{attribute 'qualified_only'}
VAR_GLOBAL
		
	//AnyEstopPressed 			: BOOL;
	//AllDCpsuOK					: BOOL;
	//AnyChargerOverTemp			: BOOL;
	//AnyChargerLoadFault			: BOOL;
	//AnyChargerInterlockOpen		: BOOL;
	//AnyChargerFaulted			: BOOL; // same as summary fault
	
	//SystemTripped 				: BOOL;
	//InstrumentationFaulted		: BOOL;
	//AnyChargeRlyFail			: BOOL;
	//AnyDumpRlyFail				: BOOL;
	//AnyACInterlockFail			: BOOL;
	//AnyLossInhibitSignal		: BOOL;
	//AnyLossHVONsignal			: BOOL;
	
	ChargingTimerRunout         : BOOL;
	ChargedTimerRunout			: BOOL;
	DumpTimerRunout				: BOOL;
	//SystemTimeOut				: BOOL;
	NoFaultDetected				: BOOL;
	TimerRunOutON				: BOOL;
	
	ChargerSummaryFault			: BOOL;
	
	EStopPBpressed				: BOOL;
	CageDoorNotClose			: BOOL;
	ShortingSystemUnknown		: BOOL;
END_VAR

(* stored: Version 1.1.0.1, ProductVersion 3.1.4024.11
   GVL Trips_DB: Id {b9292f11-9c83-43f6-9b30-6c69cf4aaa02} *)
